TYPE ST_Fenster_Parameter :
STRUCT
	Zeit_Stellen1			: DINT;
	Zeit_Stellen0			: DINT;

	AutoQuittierung			: BOOL;
END_STRUCT
END_TYPE

(* stored: Version 1.1.0.1, ProductVersion 3.1.4024.9
   DUT ST_Fenster_Parameter: Id {e25c2723-7e1d-4bdb-9a3b-ab612f8c2024} *)
